# EPICS substitutions: ThingyApp/Db/notifyNumber.substitutions
file "notifyNumber.template" {

# PV name is $(Sys)$(Dev)$(Attr)

pattern { Sys,	Dev,			Attr,			Units,		NodeID,	SensorID}

{ "XF:10IDB",	"{THINGY:BRIDGE}","Battery"	,	"%",		10,		0}

{ "XF:10IDB",	"{THINGY:001}",	"Battery"	,	"%",		0,		0}
{ "XF:10IDB",	"{THINGY:001}",	"Temperature",	"C",		0,		1}
{ "XF:10IDB",	"{THINGY:001}",	"Humidity",		"%",		0,		2}
{ "XF:10IDB",	"{THINGY:001}",	"Pressure",		"hPa",		0,		3}

{ "XF:10IDB",	"{THINGY:002}",	"Battery"	,	"%",		1,		0}
{ "XF:10IDB",	"{THINGY:002}",	"Temperature",	"C",		1,		1}
{ "XF:10IDB",	"{THINGY:002}",	"Humidity",		"%",		1,		2}
{ "XF:10IDB",	"{THINGY:002}",	"Pressure",		"hPa",		1,		3}

{ "XF:10IDB",	"{THINGY:003}",	"Battery"	,	"%",		2,		0}
{ "XF:10IDB",	"{THINGY:003}",	"Temperature",	"C",		2,		1}
{ "XF:10IDB",	"{THINGY:003}",	"Humidity",		"%",		2,		2}
{ "XF:10IDB",	"{THINGY:003}",	"Pressure",		"hPa",		2,		3}

{ "XF:10IDB",	"{THINGY:004}",	"Battery"	,	"%",		3,		0}
{ "XF:10IDB",	"{THINGY:004}",	"Temperature",	"C",		3,		1}
{ "XF:10IDB",	"{THINGY:004}",	"Humidity",		"%",		3,		2}
{ "XF:10IDB",	"{THINGY:004}",	"Pressure",		"hPa",		3,		3}

}
